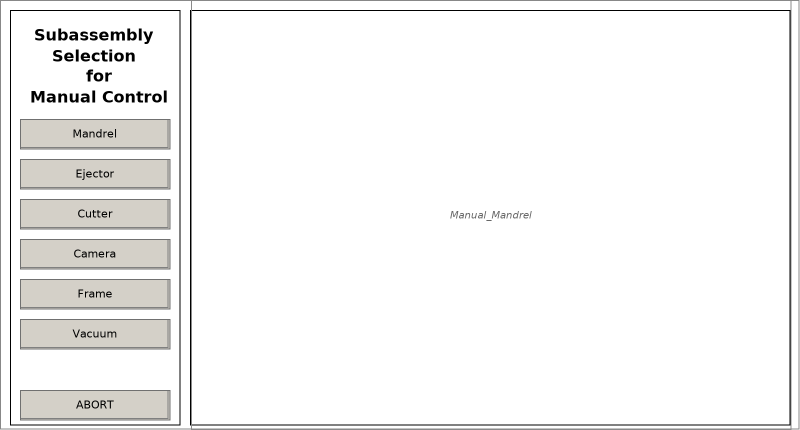
VISUALIZATION ManualControl  // 800x430
    Rectangle (190,10 600x415)
    Frame (191,0 600x430)
        shows Manual_Mandrel()
        shows Manual_Ejector()
        shows Manual_Cutter()
        shows Manual_Camera()
        shows Manual_Frame()
        shows Manual_Select_Tube()
        shows Manual_Vacuum()
    Rectangle (10,10 170x415)
    Button (20,119 150x30), "Mandrel"
        OnMouseClick: FrameSelectionChange Selection=SelectedFrame=b6e51242-079a-4729-85ea-e161656839df, GlobSel=AssignType=Directly, SelType=Locally
        OnMouseClick: execute { MAIN.TubeHmi := Main.Tube; }
    Button (20,159 150x30), "Ejector"
        OnMouseClick: FrameSelectionChange Selection=SelectedFrame=b6e51242-079a-4729-85ea-e161656839df, Selection=1, GlobSel=AssignType=Directly, SelType=Locally
    Button (20,199 150x30), "Cutter"
        OnMouseClick: FrameSelectionChange Selection=SelectedFrame=b6e51242-079a-4729-85ea-e161656839df, Selection=2, GlobSel=AssignType=Directly, SelType=Locally
    Button (20,239 150x30), "Camera"
        OnMouseClick: FrameSelectionChange Selection=SelectedFrame=b6e51242-079a-4729-85ea-e161656839df, Selection=3, GlobSel=AssignType=Directly, SelType=Locally
    Button (20,279 150x30), "Frame"
        OnMouseClick: FrameSelectionChange Selection=SelectedFrame=b6e51242-079a-4729-85ea-e161656839df, Selection=4, GlobSel=AssignType=Directly, SelType=Locally
    Button (20,390 150x30), "ABORT"
        OnMouseClick: execute { MAIN.eCommand := E_PMLCommand.ePMLCommand_Abort; }
    Group (10,20 170x92)
        Group (0,0 170x51)
            Label (0,21 168x30), "Selection"
            Label (0,0 168x30), "Subassembly"
        Label (4,62 170x30), "Manual Control"
        Label (4,41 170x30), "for"
    Button (20,319 150x30), "Vacuum"
        OnMouseClick: FrameSelectionChange Selection=SelectedFrame=b6e51242-079a-4729-85ea-e161656839df, Selection=6, GlobSel=AssignType=Directly, SelType=Locally
END_VISUALIZATION

(* stored: Version 1.1.0.1, ProductVersion 3.1.4024.9
   Visu ManualControl: Id {1e3750d0-d333-468d-b2e0-7e435a3c1a45} *)
